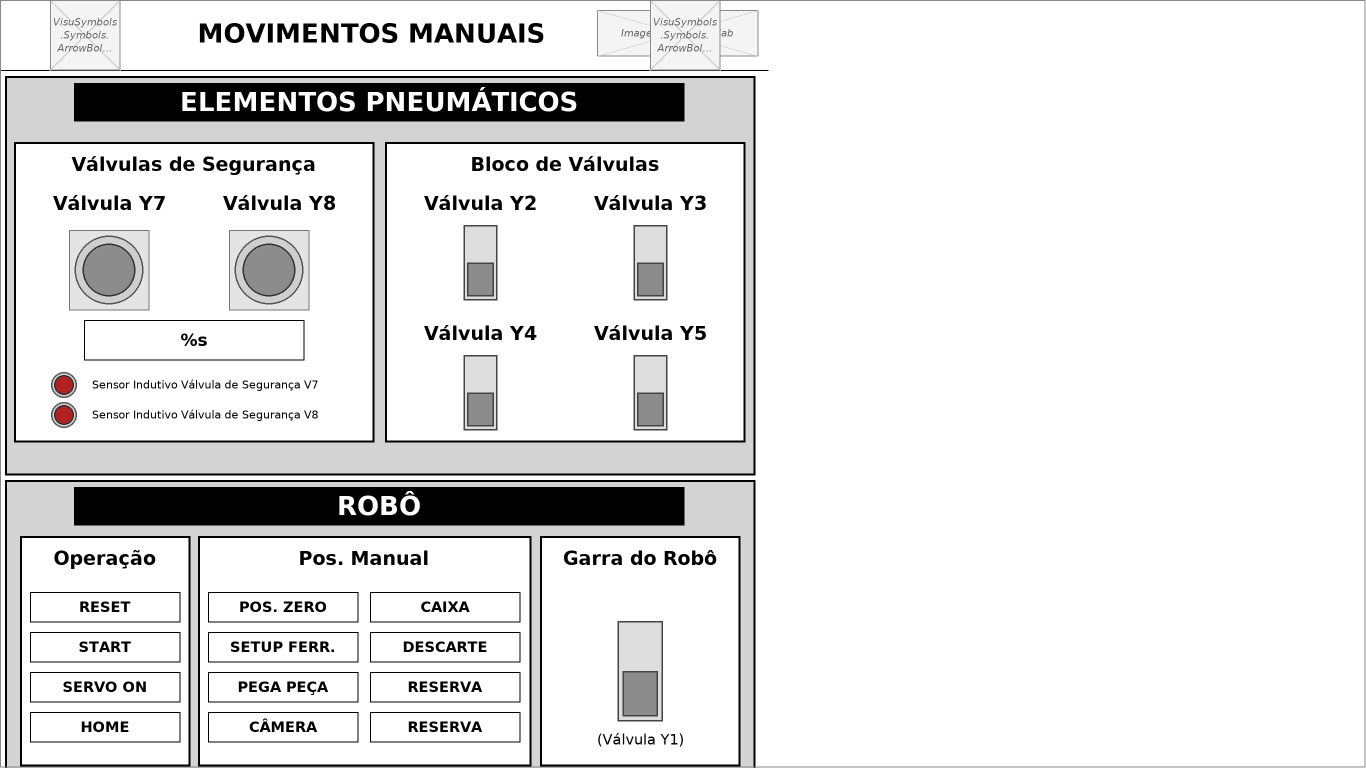
VISUALIZATION Tela_Manual_2  // 1366x768
    Group (5,480 750x305)
        RoundedRectangle (0,0 750x305)
        Rectangle (69,7 610x38), "ROBÔ", text variable: Recipe_name_Select, input disabled if: TRUE
        RoundedRectangle (15,56 170x230), input disabled if: TRUE
        Rectangle (20,65 160x27), "Operação", text variable: Recipe_name_Select, input disabled if: TRUE
        RoundedRectangle (25,112 150x30), "RESET", input disabled if: TRUE
            tap Servos.ResetServoX
        RoundedRectangle (25,152 150x30), "START", colour toggle: NOT Servos.PowerOnServoX, input disabled if: TRUE
        RoundedRectangle (193,56 333x230), input disabled if: TRUE
        Rectangle (279,65 160x27), "Pos. Manual", text variable: Recipe_name_Select, input disabled if: TRUE
        RoundedRectangle (203,112 150x30), "POS. ZERO", input disabled if: TRUE
        RoundedRectangle (203,152 150x30), "SETUP FERR.", colour toggle: NOT Servos.PowerOnServoX, input disabled if: TRUE
        RoundedRectangle (203,192 150x30), "PEGA PEÇA", colour toggle: NOT Servos.PowerOnServoX, input disabled if: TRUE
        RoundedRectangle (203,232 150x30), "CÂMERA", colour toggle: NOT Servos.PowerOnServoX, input disabled if: TRUE
        RoundedRectangle (535,56 200x230), input disabled if: TRUE
        Rectangle (545,65 180x27), "Garra do Robô", text variable: Recipe_name_Select, input disabled if: TRUE
        RoundedRectangle (25,232 150x30), "HOME", colour toggle: NOT Servos.PowerOnServoX, input disabled if: TRUE
        RoundedRectangle (25,192 150x30), "SERVO ON", input disabled if: TRUE
            tap Servos.ResetServoX
        DipSwitch (585,141 100x100), variable: IhmBt_Y1_Ligar, input disabled if: NOT MaquinaModoManual, behaviour: TOGGLE, style: Switch-DipSwitch-Gray
        Rectangle (578,246 115x27), "(Válvula Y1)", text variable: Recipe_name_Select, input disabled if: TRUE
        RoundedRectangle (365,232 150x30), "RESERVA", colour toggle: NOT Servos.PowerOnServoX, input disabled if: TRUE
        RoundedRectangle (365,112 150x30), "CAIXA", input disabled if: TRUE
        RoundedRectangle (365,152 150x30), "DESCARTE", colour toggle: NOT Servos.PowerOnServoX, input disabled if: TRUE
        RoundedRectangle (365,192 150x30), "RESERVA", colour toggle: NOT Servos.PowerOnServoX, input disabled if: TRUE
    Line (0,70) (768,70)
    Line (0,1312) (768,1312)
    Image (597,10 161x46), image: ImagePool.Logo_Indab
    Rectangle (584,1340 180x24), "%t[dd/MM/yyyy]"
    Rectangle (584,1316 180x24), "%t[HH:mm:ss]"
    Label (153,7 437x53), "MOVIMENTOS MANUAIS"
    Button (15,1315 175x45), "RECEITAS"
        OnMouseClick: change screen: Tela_Receita
    Button (375,1315 175x45), "MANUTENÇÃO"
        OnMouseClick: change screen: Tela_Manutencao
    Image (50,0 70x70), image: VisuSymbols.Symbols.ArrowBoldLeft
        OnMouseClick: change screen: Tela_Manual_1
    Image (650,0 70x70), image: VisuSymbols.Symbols.ArrowBoldRight
        OnMouseClick: change screen: Tela_Manual_3
    Button (195,1315 175x45), "PRODUÇÃO"
        OnMouseClick: change screen: Tela_Producao
    RoundedRectangle (5,76 750x399)
    Rectangle (74,83 610x38), "ELEMENTOS PNEUMÁTICOS", text variable: Recipe_name_Select
    RoundedRectangle (385,142 360x300), input disabled if: NOT MaquinaModoManual
    Rectangle (399,151 332x27), "Bloco de Válvulas", text variable: Recipe_name_Select, input disabled if: NOT MaquinaModoManual
    RoundedRectangle (14,142 360x300), input disabled if: NOT MaquinaModoManual
    Rectangle (28,151 332x27), "Válvulas de Segurança", text variable: Recipe_name_Select, input disabled if: NOT MaquinaModoManual
    Rectangle (52,190 115x27), "Válvula Y7", text variable: Recipe_name_Select, input disabled if: TRUE
    Rectangle (222,190 115x27), "Válvula Y8", text variable: Recipe_name_Select, input disabled if: TRUE
    PushSwitchLed (69,230 80x80), variable: IhmBt_Y7_Ligar, input disabled if: TRUE, behaviour: TOGGLE, style: Switch-PushSwitchLed-Gray
    PushSwitchLed (229,230 80x80), variable: IhmBt_Y8_Ligar, input disabled if: TRUE, behaviour: TOGGLE, style: Switch-PushSwitchLed-Gray
    Rectangle (423,190 115x27), "Válvula Y2", text variable: Recipe_name_Select, input disabled if: NOT MaquinaModoManual
    Rectangle (593,190 115x27), "Válvula Y3", text variable: Recipe_name_Select, input disabled if: NOT MaquinaModoManual
    DipSwitch (443,225 75x75), variable: IhmBt_Y2_Ligar, input disabled if: NOT MaquinaModoManual, behaviour: TOGGLE, style: Switch-DipSwitch-Gray
    DipSwitch (613,225 75x75), variable: IhmBt_Y3_Ligar, input disabled if: NOT MaquinaModoManual, behaviour: TOGGLE, style: Switch-DipSwitch-Gray
    Rectangle (423,320 115x27), "Válvula Y4", text variable: Recipe_name_Select, input disabled if: NOT MaquinaModoManual
    Rectangle (593,320 115x27), "Válvula Y5", text variable: Recipe_name_Select, input disabled if: NOT MaquinaModoManual
    DipSwitch (613,355 75x75), variable: IhmBt_Y5_Ligar, input disabled if: NOT MaquinaModoManual, behaviour: TOGGLE, style: Switch-DipSwitch-Gray
    DipSwitch (443,355 75x75), variable: IhmBt_Y4_Ligar, input disabled if: NOT MaquinaModoManual, behaviour: TOGGLE, style: Switch-DipSwitch-Gray
    Rectangle (84,320 220x40), "%s", text variable: IhmVs_PressaoPainelPneumatico_Text, colour toggle: Alarmes.ByteAlarmePainelPneumatico.0, input disabled if: NOT MaquinaModoManual
    Group (49,370 290x60), input disabled if: NOT MaquinaModoManual
        Rectangle (40,30 250x30), "Sensor Indutivo Válvula de Segurança V8"
        Lamp1 (0,0 30x30), variable: Alarmes.ByteAlarmePainelPneumatico.1, style: Lamp-Lamp1-Red
        Rectangle (40,0 250x30), "Sensor Indutivo Válvula de Segurança V7"
        Lamp1 (0,30 30x30), variable: Alarmes.ByteAlarmePainelPneumatico.2, style: Lamp-Lamp1-Red
    Line (-1,1315) (767,1315)
    RoundedRectangle (5,790 750x511)
    Rectangle (75,800 610x38), "MOTORES", text variable: Recipe_name_Select, input disabled if: NOT MaquinaModoManual
    Button (260,1235 240x60), "MODO: %s", text variable: IhmBt_ManualAuto_Text, colour toggle: IhmBt_ManualAuto_Color
        toggle IhmBt_ManualAuto
    RoundedRectangle (24,855 350x360), input disabled if: NOT MaquinaModoManual
    Rectangle (146,863 106x27), "Servo X", text variable: Recipe_name_Select, input disabled if: NOT MaquinaModoManual
    Rectangle (31,895 77x22), "Posição", input disabled if: NOT MaquinaModoManual
    Rectangle (106,895 90x22), "%.2f mm", text variable: IhmLeit_ServoX_Posicao, input disabled if: NOT MaquinaModoManual
    RoundedRectangle (38,1165 150x30), "REFERENCIAR", input disabled if: NOT MaquinaModoManual
        tap IhmBt_ServoX_Referenciar
    RoundedRectangle (38,1125 150x30), "POWER ON", input disabled if: NOT MaquinaModoManual
        toggle IhmBt_ServoX_PowerOn
    RoundedRectangle (38,1025 150x30), "HOME", colour toggle: NOT Servos.PowerOnServoX, input disabled if: NOT MaquinaModoManual
        tap IhmBt_ServoX_Home
    RoundedRectangle (38,985 150x30), "RESET", input disabled if: NOT MaquinaModoManual
        tap IhmBt_ServoX_Reset
    Image (38,1065 50x50), invisible if: NOT IhmBt_ServoX_PowerOn, input disabled if: NOT MaquinaModoManual, image: VisuSymbols.Symbols.ArrowBoldLeft
        OnMouseDown: execute { IhmBt_ServoX_JogBwd := TRUE; }
        OnMouseLeave: execute { IhmBt_ServoX_JogBwd := FALSE; }
        OnMouseUp: execute { IhmBt_ServoX_JogBwd := FALSE; }
    Image (138,1065 50x50), invisible if: NOT IhmBt_ServoX_PowerOn, input disabled if: NOT MaquinaModoManual, image: VisuSymbols.Symbols.ArrowBoldRight
        OnMouseDown: execute { IhmBt_ServoX_JogFwd := TRUE; }
        OnMouseLeave: execute { IhmBt_ServoX_JogFwd := FALSE; }
        OnMouseUp: execute { IhmBt_ServoX_JogFwd := FALSE; }
    Rectangle (90,1079 45x20), "JOG", invisible if: NOT IhmBt_ServoX_PowerOn, input disabled if: NOT MaquinaModoManual
    Rectangle (31,920 77x22), "Velocidade:", input disabled if: NOT MaquinaModoManual
    Rectangle (106,920 90x22), "%.2f mm/s", text variable: IhmLeit_ServoX_Velocidade, input disabled if: NOT MaquinaModoManual
    Rectangle (31,945 77x22), "Torque:", input disabled if: NOT MaquinaModoManual
    Rectangle (106,945 90x22), "%d kgfm", text variable: IhmLeit_ServoX_Torque, input disabled if: NOT MaquinaModoManual
    RoundedRectangle (384,855 350x360), input disabled if: NOT MaquinaModoManual
    Rectangle (506,864 106x27), "Servo Y", text variable: Recipe_name_Select, input disabled if: NOT MaquinaModoManual
    RoundedRectangle (398,1165 150x30), "REFERENCIAR", input disabled if: NOT MaquinaModoManual
        tap IhmBt_ServoY_Referenciar
    RoundedRectangle (398,1125 150x30), "POWER ON", input disabled if: NOT MaquinaModoManual
        toggle IhmBt_ServoY_PowerOn
    RoundedRectangle (398,1025 150x30), "HOME", colour toggle: NOT Servos.PowerOnServoX, input disabled if: NOT MaquinaModoManual
        tap IhmBt_ServoY_Home
    RoundedRectangle (398,985 150x30), "RESET", input disabled if: NOT MaquinaModoManual
        tap IhmBt_ServoY_Reset
    Image (398,1065 50x50), invisible if: NOT IhmBt_ServoY_PowerOn, input disabled if: NOT MaquinaModoManual, image: VisuSymbols.Symbols.ArrowBoldLeft
        OnMouseDown: execute { IhmBt_ServoY_JogBwd := TRUE; }
        OnMouseLeave: execute { IhmBt_ServoY_JogBwd := FALSE; }
        OnMouseUp: execute { IhmBt_ServoY_JogBwd := FALSE; }
    Image (498,1065 50x50), invisible if: NOT IhmBt_ServoY_PowerOn, input disabled if: NOT MaquinaModoManual, image: VisuSymbols.Symbols.ArrowBoldRight
        OnMouseDown: execute { IhmBt_ServoY_JogFwd := TRUE; }
        OnMouseLeave: execute { IhmBt_ServoY_JogFwd := FALSE; }
        OnMouseUp: execute { IhmBt_ServoY_JogFwd := FALSE; }
    Rectangle (450,1079 45x20), "JOG", text variable: Recipe_name_Select, invisible if: NOT IhmBt_ServoY_PowerOn, input disabled if: NOT MaquinaModoManual
    Rectangle (391,895 77x22), "Posição", input disabled if: NOT MaquinaModoManual
    Rectangle (391,920 77x22), "Velocidade:", input disabled if: NOT MaquinaModoManual
    Rectangle (391,945 77x22), "Torque:", input disabled if: NOT MaquinaModoManual
    Rectangle (466,945 90x22), "%d kgfm", text variable: IhmLeit_ServoY_Torque, input disabled if: NOT MaquinaModoManual
    Rectangle (466,895 90x22), "%.2f mm", text variable: IhmLeit_ServoY_Posicao, input disabled if: NOT MaquinaModoManual
    Rectangle (466,920 90x22), "%.2f mm/s", text variable: IhmLeit_ServoY_Velocidade, input disabled if: NOT MaquinaModoManual
    RoundedRectangle (210,915 150x30), "INICIO DE CURSO", input disabled if: MaquinaModoAuto OR NOT IhmBt_ServoX_PowerOn
        toggle IhmBt_ServoX_ReferenciarAutoINICIO
    Rectangle (220,1125 130x30), "(Sensor Fim de Curso)"
    Lamp1 (270,955 30x30), variable: InFimCurso3, style: Lamp-Lamp1-Red
    Rectangle (220,985 130x30), "(Sensor Fim de Curso)"
    Lamp1 (270,1095 30x30), variable: InFimCurso4, style: Lamp-Lamp1-Red
    RoundedRectangle (210,1055 150x30), "FIM DE CURSO", input disabled if: MaquinaModoAuto OR NOT IhmBt_ServoX_PowerOn
        toggle IhmBt_ServoX_ReferenciarAutoFIM
    RoundedRectangle (570,915 150x30), "INICIO DE CURSO", input disabled if: MaquinaModoAuto OR NOT IhmBt_ServoY_PowerOn
        toggle IhmBt_ServoY_ReferenciarAutoINICIO
    Lamp1 (630,955 30x30), variable: InFimCurso1, style: Lamp-Lamp1-Red
    Rectangle (580,1125 130x30), "(Sensor Fim de Curso)"
    Rectangle (580,985 130x30), "(Sensor Fim de Curso)"
    Lamp1 (630,1095 30x30), variable: InFimCurso2, style: Lamp-Lamp1-Red
    RoundedRectangle (570,1055 150x30), "FIM DE CURSO", input disabled if: MaquinaModoAuto OR NOT IhmBt_ServoY_PowerOn
        toggle IhmBt_ServoY_ReferenciarAutoFIM
END_VISUALIZATION

(* stored: Version 1.1.0.1, ProductVersion 3.1.4024.11
   Visu Tela_Manual_2: Id {e4576a75-0062-4923-865f-b821bdd719c0} *)
